(* IEC 61131-3 sources: Industry-PLC-LLM/data/PLCBEAD_repo/PLCBEAD_PLCEmbed-main/PLC-BEAD/Source/GEB/Network_MB_SERVER, 1 file *)

(* ---- MB_SERVER.ST ---- *)
TYPE
	oscat_IP_FIFO128_DATA  : ARRAY [1..128] OF BYTE;
	oscat_Mailbox  : ARRAY [1..16] OF BYTE;

	oscat_NW_BUF_SHORT : ARRAY [0..1407] OF BYTE;
	oscat_NW_BUF_LONG  : ARRAY [0..4095] OF BYTE;

	oscat_IP_FIFO_DATA :
	STRUCT
		X       : oscat_IP_FIFO128_DATA; (* IP_ID FIFO Speicher          *)
		Y       : oscat_IP_FIFO128_DATA; (* IP_ID Z�hler                 *)
		ID      : BYTE;                  (* h�chste vergabene id         *)
		MAX_ID  : BYTE;                  (* maximal Anmeldungen pro ID   *)
		INIT    : BOOL;                  (* Initialisierung durchgef�hrt *)
		EMPTY   : BOOL;                  (* FIFO leer                    *)
		FULL    : BOOL;                  (* FIFO voll                    *)
		TOP     : INT;                   (* maximale anzahl IN FIFO      *)
		NW      : INT;                   (* Schreibzeiger                *)
		NR      : INT;                   (* Lesezeiger                   *)
	END_STRUCT;

	oscat_IP_C:
	STRUCT
		C_MODE:			BYTE;          		(*W Mode: TCP/UCP AKTIV/PASSIV                               *)
		C_PORT:         WORD;          		(*W Portnummer                                               *)
		C_IP:           DWORD;         		(*W IP-ADRESSe gepackt wwxxyyzz = www.xxx.yyy.zzz            *)
		C_STATE:        BYTE;          		(*R VerbindungsSTATUS ON/OFF + Flanke ON/OFF                 *)
		C_ENABLE:       BOOL;          		(*W Freigabe f�r Connect                                     *)
		R_OBSERVE:      BOOL;          		(*W Empfang ueberwachen                                      *)
		TIME_RESET:     BOOL;          		(*W Alle Timer ruecksetzen                                   *)
		ERROR:          DWORD;         		(*R vvwwxxyy (vv = CON_ERROR, ww = SEN_ERROR, xx = REC_ERROR *)
		FIFO:           oscat_IP_FIFO_DATA; (*I IP FIFO Struktur                                         *)
		MAILBOX:		oscat_Mailbox;		(*I Mailbox: Datenbereich f�r Bausteindatenaustausch         *)
	END_STRUCT;

	oscat_NETWORK_BUFFER :
	STRUCT
		SIZE   : UINT;
		BUFFER : oscat_NW_BUF_LONG;
	END_STRUCT;

	oscat_NETWORK_BUFFER_SHORT :
	STRUCT
	SIZE   : UINT;
	BUFFER : oscat_NW_BUF_SHORT;
	END_STRUCT;

	oscat_aW0_255	: ARRAY [0..255] OF WORD;
	oscat_VMAP_DATA :
	STRUCT
		FC       : DWORD;
		V_ADR    : INT;
		V_SIZE   : INT;
		P_ADR    : INT;
		TIME_OUT : TIME;
	END_STRUCT;

	oscat_MB_VMAP : ARRAY [1..10] OF oscat_VMAP_DATA;

	csv_parser_demo_col : ARRAY [1..4] OF REAL;
	csv_parser_demo     : ARRAY [1..2] OF csv_parser_demo_col;

END_TYPE

FUNCTION_BLOCK MB_VMAP_Block

	VAR_IN_OUT
		VMAP :	oscat_MB_VMAP;
	END_VAR

	VAR_INPUT
		FC :	INT;
		V_ADR :	INT;
		V_CNT :	INT;
		SIZE :	INT;
	END_VAR

	VAR_OUTPUT
		P_ADR :	INT;
		P_BIT :	INT;
		ERROR :	BYTE;
	END_VAR

	VAR
		i :	INT;
		VOPT :	DWORD;
		vadr :	INT;
		padr :	INT;
		mask :	DWORD;
		VSIZE :	INT;
		w_tmp :	WORD;
		i_tmp :	INT;
		init :	BOOL;
	END_VAR

	IF init = FALSE THEN
		init := TRUE;
		IF VMAP[1].FC = DWORD#0 THEN
			VMAP[1].FC := DWORD#16#FFFF_FFFF;
			VMAP[1].V_ADR := 0;
			VMAP[1].V_SIZE := 256;
			VMAP[1].P_ADR := 0;
		END_IF;
	END_IF;

	ERROR := BYTE#02;
	mask := SHL(DWORD#1,FC);

	IF (mask AND DWORD#2#00000000_01000000_00000000_01100000) <> DWORD#0 THEN
		V_CNT := 1;
	ELSIF V_CNT = 0 THEN
		RETURN;
	END_IF;

	FOR i := 1 TO 10 DO
		VOPT := VMAP[i].FC;
		IF (VOPT AND mask) <> DWORD#0 THEN
			vadr := VMAP[i].V_ADR;
			VSIZE := VMAP[i].V_SIZE;
			padr := VMAP[i].P_ADR;

			IF (mask AND DWORD#2#00000000_00000000_10000000_00100110) <> DWORD#0 THEN
				i_tmp := WORD_TO_INT(SHR(INT_TO_WORD(V_ADR + V_CNT -1),4))+1;
				IF i_tmp <= SIZE AND i_tmp <= VSIZE THEN
					w_tmp := INT_TO_WORD(V_ADR);
					P_ADR := WORD_TO_INT(SHR(w_tmp,4)) + padr;
					P_BIT := WORD_TO_INT(w_tmp AND WORD#16#000F);
					ERROR := BYTE#0;
					EXIT;
				END_IF;
			ELSIF (mask AND DWORD#2#00000000_11000001_00000000_01011000) <> DWORD#0 THEN
				IF V_ADR >= vadr AND V_ADR + V_CNT <= vadr + VSIZE THEN
					P_ADR := V_ADR - vadr + padr;
					IF P_ADR + V_CNT <= SIZE THEN
						ERROR := BYTE#0;
						EXIT;
					END_IF;
				END_IF;
			ELSE
				ERROR := BYTE#01;
				RETURN;
			END_IF;
		END_IF;
	END_FOR;

	IF ERROR = BYTE#0 THEN
		IF (mask AND DWORD#2#00000000_11000001_10000000_01100000) <> DWORD#0 THEN
			VMAP[i].TIME_OUT := T#1ms;
		END_IF;
	END_IF;

END_FUNCTION_BLOCK

FUNCTION _BYTE_TO_INT:INT
	VAR_INPUT
		IN :	BYTE;
	END_VAR

	_BYTE_TO_INT := USINT_TO_INT(BYTE_TO_USINT(IN));
END_FUNCTION

FUNCTION_BLOCK IP_FIFO_Block

  VAR_IN_OUT
    FIFO :	oscat_IP_FIFO_DATA;
    ID :	BYTE;
    STATE :	BYTE;
  END_VAR

  VAR
    tmp :	INT;
  END_VAR

  IF NOT FIFO.INIT THEN
    FIFO.INIT		:= TRUE;
    FIFO.NW		:= 1;
    FIFO.NR		:= 1;
    FIFO.EMPTY	:= TRUE;
    FIFO.FULL		:= FALSE;
    FIFO.TOP		:= 128;
    FIFO.MAX_ID	:= BYTE#1;
  END_IF;

  IF ID = BYTE#00 THEN
    IF FIFO.ID < INT_TO_BYTE(FIFO.TOP) THEN
      ID := USINT_TO_BYTE(BYTE_TO_USINT(FIFO.ID) + USINT#1);
      FIFO.ID := ID ;

    ELSIF STATE < BYTE#200 THEN
      STATE := BYTE#255;
    RETURN;
    END_IF;
  END_IF;

  IF STATE = BYTE#1 AND NOT FIFO.FULL THEN
    tmp := _BYTE_TO_INT(ID);
    IF FIFO.Y[tmp] < FIFO.MAX_ID THEN
      FIFO.Y[tmp] := USINT_TO_BYTE(BYTE_TO_USINT(FIFO.Y[tmp]) + USINT#1);
      tmp := FIFO.NW;
      FIFO.X[tmp] := ID;
      IF FIFO.NW = FIFO.TOP THEN FIFO.NW := 1; ELSE FIFO.NW := FIFO.NW + 1; END_IF;
      FIFO.FULL := FIFO.NW = FIFO.NR;
    FIFO.EMPTY := FALSE;
      STATE := BYTE#2;
    END_IF;
  END_IF;

  IF STATE = BYTE#2 AND NOT FIFO.EMPTY THEN
    tmp := FIFO.NR;
    IF ID = FIFO.X[tmp] THEN
      STATE := BYTE#3;
    END_IF;
  END_IF;

  IF STATE = BYTE#4 AND NOT FIFO.EMPTY THEN

    tmp := FIFO.NR;
    IF ID = FIFO.X[tmp] THEN
      tmp := _BYTE_TO_INT(ID);
      FIFO.Y[tmp] := USINT_TO_BYTE(BYTE_TO_USINT(FIFO.Y[tmp]) - USINT#1);

      IF FIFO.NR = FIFO.TOP THEN FIFO.NR := 1; ELSE FIFO.NR := FIFO.NR + 1; END_IF;
      FIFO.EMPTY := FIFO.NR = FIFO.NW;
    FIFO.FULL := FALSE;
    END_IF;
    STATE := BYTE#5;
  END_IF;

END_FUNCTION_BLOCK

FUNCTION _UDINT_TO_TIME:TIME

	VAR_INPUT
		IN :	UDINT;
	END_VAR

	_UDINT_TO_TIME := DINT_TO_TIME(UDINT_TO_DINT(IN));

END_FUNCTION

FUNCTION_BLOCK T_PLC_MS_block

	VAR_OUTPUT
		T_PLC_MS :	UDINT;
	END_VAR

	VAR
		PLC_TICKS_PER_SEC :	INT;
		PLC_SYS_TICK_CNT :	DINT;
	END_VAR

	VAR
		debug :	BOOL;(*Debug-Mode ON / OFF*)
		N :	INT;(*Debug-Faktor*)
		Offset :	UDINT;(*Debug-Offset*)
		temp :	DWORD := DWORD#1;(*Debug-Offset*)
		MODE :	BOOL;(*modus*)
		faktor :	UDINT;(*Systemtakt-Faktor*)
		init :	BOOL;
		v_plc_ticks_per_sec :	UDINT;
		base :	UDINT := UDINT#1000;
	END_VAR

	IF init = FALSE THEN
		v_plc_ticks_per_sec := INT_TO_UDINT(PLC_TICKS_PER_SEC);
		IF v_plc_ticks_per_sec = UDINT#1024 THEN
			faktor := UDINT#1;
			MODE := FALSE;
		ELSIF v_plc_ticks_per_sec > UDINT#0 THEN
			IF v_plc_ticks_per_sec <= base THEN
				faktor := base / v_plc_ticks_per_sec;
				MODE := FALSE;
			ELSE
				faktor := v_plc_ticks_per_sec / base;
				MODE := TRUE;
			END_IF;
		ELSE
			faktor := UDINT#1;
		END_IF;
		init := TRUE;
	END_IF;

	IF MODE THEN
		T_PLC_MS := DINT_TO_UDINT(PLC_SYS_TICK_CNT) / faktor;
	ELSE
		T_PLC_MS := DINT_TO_UDINT(PLC_SYS_TICK_CNT) * faktor;
	END_IF;

	IF debug THEN
		T_PLC_MS := (DWORD_TO_UDINT(SHL(UDINT_TO_DWORD(T_PLC_MS),N) OR SHL(temp,N)) - UDINT#1) + Offset;
	END_IF;

END_FUNCTION_BLOCK

FUNCTION WORD_OF_BYTE:WORD
	VAR_INPUT
		B1 :	BYTE;
		B0 :	BYTE;
	END_VAR
	WORD_OF_BYTE := SHL(BYTE_TO_WORD(B1),8) OR BYTE_TO_WORD(B0);
END_FUNCTION

FUNCTION BIT_LOAD_W:WORD
	VAR_INPUT
		IN :	WORD;
		VAL :	BOOL;
		POS :	INT;
	END_VAR

	IF VAL THEN
		BIT_LOAD_W := IN OR SHL(WORD#1,POS);
	ELSE
		BIT_LOAD_W := IN AND (NOT SHL(WORD#1,POS));
	END_IF;
END_FUNCTION

FUNCTION_BLOCK MB_SERVER_Block

	VAR_IN_OUT
		IP_C :	oscat_IP_C;
		S_BUF :	oscat_NETWORK_BUFFER_SHORT;
		R_BUF :	oscat_NETWORK_BUFFER_SHORT;
		VMAP :	oscat_MB_VMAP;
		DATA :	oscat_aW0_255;
	END_VAR

	VAR_INPUT
		DATA_SIZE :	INT;
		ENABLE :	BOOL;
		UDP :	BOOL;
	END_VAR

	VAR_OUTPUT
		ERROR :	DWORD;
	END_VAR

	VAR
		MB_VMAP :	MB_VMAP_Block;
		adR1  :	INT;
		adR2 :	INT;
		points :	INT;
		pointS2 :	INT;
		coils :	BYTE;
		mask :	BYTE;
		idX1 :	INT;
		idX2 :	INT;
		BIT_POS :	INT;
		count :	INT;
		fc :	INT;
		i :	INT;
		STATE :	INT;
		IP_STATE :	BYTE;
		IP_ID :	BYTE;
		IP_FIFO :	IP_FIFO_Block;
		w_tmp :	WORD;
		last_cycle :	TIME;
		TX :	TIME;
		T_PLC_MS :	T_PLC_MS_block;
		t :	TON;
		ip_ERROR :	BOOL;
	END_VAR

	T_PLC_MS();
	TX := UDINT_TO_TIME(T_PLC_MS.T_PLC_MS);

	FOR i := 1 TO 10 DO
		IF VMAP[i].TIME_OUT > T#0s THEN
			VMAP[i].TIME_OUT := VMAP[i].TIME_OUT + SUB_TIME(TX, last)_cycle;
		END_IF;
	END_FOR;
	last_cycle := TX;
	ip_ERROR := IP_C.ERROR > DWORD#0;

	CASE STATE OF

	00:
		IF ENABLE THEN
			STATE := 10;
			IP_STATE := BYTE#1;
		END_IF;

	10:
		IF IP_STATE = BYTE#3 THEN

			IP_C.C_PORT     := WORD#0;
			IP_C.C_IP       := DWORD#0;
			IP_C.C_MODE     := SEL(UDP,BYTE#4,BYTE#5);
			IP_C.TIME_RESET := TRUE;
			IP_C.C_ENABLE   := TRUE;
			IP_C.R_OBSERVE  := FALSE;
			STATE := 20;
		END_IF;

	20:	IF NOT ip_ERROR THEN
			IF S_BUF.SIZE = UINT#0 AND R_BUF.SIZE > UINT#6 THEN
				IF  R_BUF.SIZE = WORD_TO_UINT(WORD_OF_BYTE(R_BUF.BUFFER[4],R_BUF.BUFFER[5])) + UINT#6 THEN
					ERROR := DWORD#00;

					FOR i := 0 TO 13 DO
						S_BUF.BUFFER[i] := R_BUF.BUFFER[i];
					END_FOR;

					fc := _BYTE_TO_INT(R_BUF.BUFFER[7]);

					adR1  := WORD_TO_INT(WORD_OF_BYTE(R_BUF.BUFFER[8],R_BUF.BUFFER[9]));
					points := WORD_TO_INT(WORD_OF_BYTE(R_BUF.BUFFER[10],R_BUF.BUFFER[11]));

					MB_VMAP(VMAP:=VMAP,FC:=fc,V_ADR:=adR1 ,V_CNT:=points,SIZE:=DATA_SIZE);
					VMAP:=MB_VMAP.VMAP;
					adR1 :=MB_VMAP.P_ADR;
					BIT_POS:=MB_VMAP.P_BIT;
					ERROR:=BYTE_TO_DWORD(MB_VMAP.ERROR);

					IF ERROR = DWORD#0 THEN
						CASE fc OF

						1..2 :
							count := 9;
							coils := BYTE#0;
							mask := BYTE#1;
							FOR i := 1 TO points DO
								IF mask = BYTE#0 THEN
									mask := BYTE#1;
									S_BUF.BUFFER[count] := coils;
									coils := BYTE#0;
									count := count + 1;
								END_IF;
								IF (DATA[adR1 ] AND SHL(WORD#1,BIT_POS)) > WORD#0 THEN
									coils := coils OR mask;
								END_IF;

								BIT_POS := BIT_POS + 1;
								IF BIT_POS > 15 THEN
									adR1  := adR1  + 1;
									BIT_POS := 0;
								END_IF;

								mask := SHL(mask,1);
							END_FOR;
							S_BUF.BUFFER[Count] := coils;

							S_BUF.BUFFER[8] := INT_TO_BYTE(count - 8);
							S_BUF.SIZE := INT_TO_UINT(count + 1);

						3..4 :
							idX1 := 07;
							count := adR1  + points - 1;
							FOR i := adR1  TO count DO
								idX1 := idX1 + 2;
								idX2 := idX1 + 1;
								w_tmp := DATA[i];
								S_BUF.BUFFER[idX1] := WORD_TO_BYTE(SHR(w_tmp,8));
								S_BUF.BUFFER[idX2] := WORD_TO_BYTE(w_tmp);
							END_FOR;
							S_BUF.BUFFER[8] := SHL(INT_TO_BYTE(points),1);
							S_BUF.SIZE := INT_TO_UINT(idX2 + 1);
						5 :
							DATA[adR1 ]:=BIT_LOAD_W(DATA[adR1 ],R_BUF.BUFFER[10]>BYTE#0,BIT_POS);
							S_BUF.SIZE := UINT#12;
						6 :
							DATA[adR1 ] := WORD_OF_BYTE(R_BUF.BUFFER[10],R_BUF.BUFFER[11]);
							S_BUF.SIZE := UINT#12;
						15 :
							mask := BYTE#1;
							idX1 := 13;
							FOR i := 1 TO points DO
								DATA[adR1 ]:=BIT_LOAD_W(DATA[adR1 ],(R_BUF.BUFFER[idX1] AND mask)>BYTE#0,BIT_POS);
								BIT_POS := BIT_POS + 1;
								IF BIT_POS > 15 THEN
									adR1  := adR1  + 1;
									BIT_POS := 0;
								END_IF;
								mask := ROL(mask,1);
								IF mask = BYTE#1 THEN
									idX1 := idX1 +1;
								END_IF;
							END_FOR;
							S_BUF.SIZE := UINT#12;
						16 :
							idX1 := 11;
							count := adR1  + points -1;
							FOR i := adR1  TO Count DO
								idX1 := idX1 + 2;
								idX2 := idX1 + 1;
								Data[i] := WORD_OF_BYTE(R_BUF.BUFFER[idX1],R_BUF.BUFFER[idX2]);
							END_FOR;
							S_BUF.SIZE := UINT#12;
						22 :
							w_tmp := WORD_OF_BYTE(R_BUF.BUFFER[11],R_BUF.BUFFER[11]);
							DATA[adR1 ] := (DATA[adR1 ] AND w_tmp) OR (WORD_OF_BYTE(R_BUF.BUFFER[12],R_BUF.BUFFER[13]) AND (NOT w_tmp));
							S_BUF.SIZE := UINT#14;
						23 :
							adR2 := WORD_TO_INT(WORD_OF_BYTE(R_BUF.BUFFER[12],R_BUF.BUFFER[13]));
							pointS2 := WORD_TO_INT(WORD_OF_BYTE(R_BUF.BUFFER[14],R_BUF.BUFFER[15]));

							MB_VMAP(VMAP:=VMAP,FC:=16,V_ADR:=adR2,V_CNT:=pointS2,SIZE:=DATA_SIZE);
							VMAP:=MB_VMAP.VMAP;
							adR2:=MB_VMAP.P_ADR;
							ERROR:=BYTE_TO_DWORD(MB_VMAP.ERROR);

							IF ERROR = DWORD#0 THEN
								idX1 := 15;
								count := adR2 + pointS2 -1;
								FOR i := adR2 TO count DO
									idX1 := idX1 + 2;
									idX2 := idX1 + 1;
									Data[i] := WORD_OF_BYTE(R_BUF.BUFFER[idX1],R_BUF.BUFFER[idX2]);
								END_FOR;

								idX1 := 07;
								count := adR1  + points - 1;
								FOR i := adR1  TO count DO
									idX1 := idX1 + 2;
									idX2 := idX1 + 1;
									w_tmp := DATA[i];
									S_BUF.BUFFER[idX1] := WORD_TO_BYTE(SHR(w_tmp,8));
									S_BUF.BUFFER[idX2] := WORD_TO_BYTE(w_tmp);
								END_FOR;
								S_BUF.BUFFER[8] := SHL(INT_TO_BYTE(points),1);
								S_BUF.SIZE := INT_TO_UINT(idX2 + 1);

							END_IF;

						ELSE
							ERROR := DWORD#01;
						END_CASE;
					END_IF;
				END_IF;

				IF ERROR > DWORD#0 THEN
					S_BUF.BUFFER[7] := S_BUF.BUFFER[7] OR BYTE#2#1000_0000;
					S_BUF.BUFFER[8] := DWORD_TO_BYTE(ERROR);
					S_BUF.SIZE := UINT#9;
				END_IF;

				S_BUF.BUFFER[4] := BYTE#0;
				S_BUF.BUFFER[5] := UINT_TO_BYTE(S_BUF.SIZE - UINT#6);

			END_IF;
		ELSE
			ERROR := IP_C.ERROR;
		END_IF;

		t(IN:= ip_ERROR, PT:=T#5s);
		IF t.Q THEN
			IP_C.TIME_RESET := TRUE;
		END_IF;

		R_BUF.SIZE := UINT#0;

		IF ENABLE = FALSE THEN
			IP_STATE := BYTE#4;
			STATE := 00;
		END_IF;
	END_CASE;

	IP_FIFO(FIFO:=IP_C.FIFO,STATE:=IP_STATE,ID:=IP_ID);
	IP_C.FIFO:=IP_FIFO.FIFO;
	IP_STATE := IP_FIFO.STATE;
	IP_ID:=IP_FIFO.ID;

END_FUNCTION_BLOCK

PROGRAM program0
	VAR
		IP_C :	oscat_IP_C;
		S_BUF :	oscat_NETWORK_BUFFER_SHORT;
		R_BUF :	oscat_NETWORK_BUFFER_SHORT;
		VMAP :	oscat_MB_VMAP;
		DATA :	oscat_aW0_255;
		DATA_SIZE :	INT;
		ENABLE :	BOOL;
		UDP :	BOOL;
		ERROR :	DWORD;

		func_block : MB_SERVER_Block;
	END_VAR
	func_block.IP_C := IP_C;
	func_block.S_BUF := S_BUF;
	func_block.R_BUF := R_BUF;
	func_block.VMAP := VMAP;
	func_block.DATA := DATA;
	func_block.DATA_SIZE := DATA_SIZE;
	func_block.ENABLE := ENABLE;
	func_block.UDP := UDP;

	func_block();
  	IP_C  := func_block.IP_C;
	S_BUF  := func_block.S_BUF;
	R_BUF  := func_block.R_BUF;
	VMAP  := func_block.VMAP;
	DATA  := func_block.DATA;
	ERROR  := func_block.ERROR;

END_PROGRAM
